FUNCTION_BLOCK EL3042
VAR
	_io : EL3xx2_Data;
	{attribute addProperty Name "WcState"}
	_wcState : WcStateInputToggle;
	{attribute addProperty Name "Info data"}
	_infoData : InfoDataAds;
END_VAR

PROPERTY IO : REFERENCE TO EL3xx2_Data
GET
IO REF= _io;
END_GET
END_PROPERTY

PROPERTY WcState : REFERENCE TO WcStateInputToggle
GET
WcState REF= _wcState;
END_GET
END_PROPERTY

END_FUNCTION_BLOCK

(* stored: Version 1.1.0.1, ProductVersion 3.1.4024.9
   POU EL3042: Id {0f35165e-9ad7-0042-0db6-622c4427422a}, SpecialFunc None
   Property IO: Id {04eedff2-7f37-024e-1bde-d46453070e4f}
   Get Get: Id {08be5bf8-a095-0b30-316e-705a2c138b69}
   Property WcState: Id {48c53a0d-277c-0827-12bc-017002dcf7c5}
   Get Get: Id {509a690a-6e10-0cd2-05dc-5795de7c556f} *)
